// SIMATIC STEP 7 (V5.x) project zEn01_13_STEP7__PID-Temp
// program: Step controller
// program: Pulse controller
// program: Pulse control OB35, OB32
// program: Pulse control OB35, OB1
// program: Continuous controller

SYMBOL_TABLE
"DB_TCONT_S"	DB 59	FB 59
"DB_PROC_S"	DB 101	FB 101
"TCONT_S"	FB 59	FB 59	// temperature PID step controller
"PROC_S"	FB 101	FB 101
"CYC_INT5"	OB 35	OB 35
"COMPLETE_RESTART"	OB 100	OB 100
"VAT_LoopControlS"	VAT 1	
END_SYMBOL_TABLE

// FB 59: know-how protected block, not included

// FB 101: know-how protected block, not included

DATA_BLOCK "DB_TCONT_S"	// DB 59
VERSION : 0.0
"TCONT_S"
BEGIN
END_DATA_BLOCK

DATA_BLOCK "DB_PROC_S"	// DB 101
VERSION : 0.0
"PROC_S"
BEGIN
END_DATA_BLOCK

ORGANIZATION_BLOCK "CYC_INT5"	// OB 35
TITLE = "Cyclic Interrupt"
VERSION : 0.1
VAR_TEMP
  OB35_EV_CLASS : BYTE ;	//Bits 0-3 = 1 (Coming event), Bits 4-7 = 1 (Event class 1)
  OB35_STRT_INF : BYTE ;	//16#36 (OB 35 has started)
  OB35_PRIORITY : BYTE ;	//11 (Priority of 1 is lowest)
  OB35_OB_NUMBR : BYTE ;	//35 (Organization block 35, OB35)
  OB35_RESERVED_1 : BYTE ;	//Reserved for system
  OB35_RESERVED_2 : BYTE ;	//Reserved for system
  OB35_PHASE_OFFSET : WORD ;	//Phase offset (msec)
  OB35_RESERVED_3 : INT ;	//Reserved for system
  OB35_EXC_FREQ : INT ;	//Frequency of execution (msec)
  OB35_DATE_TIME : DATE_AND_TIME ;	//Date and time OB35 started
END_VAR
BEGIN
NETWORK
TITLE =
//Call the controller and the simulated process
      CALL  "TCONT_S" , "DB_TCONT_S" (
           DIX 18.0                 := DB101.DBX 50.0,
           DIX 18.1                 := DB101.DBX 50.1);
      CALL  "PROC_S" , "DB_PROC_S" (
           DIX 0.0                  := DB59.DBX 20.0,
           DIX 0.1                  := DB59.DBX 20.1,
           DID 42                   := DB59.DBD 8);
END_ORGANIZATION_BLOCK

ORGANIZATION_BLOCK "COMPLETE_RESTART"	// OB 100
TITLE = "Complete Restart"
VERSION : 0.1
VAR_TEMP
  OB100_EV_CLASS : BYTE ;	//16#13, Event class 1, Entering event state, Event logged in diagnostic buffer
  OB100_STRTUP : BYTE ;	//16#81/82/83/84 Method of startup
  OB100_PRIORITY : BYTE ;	//27 (Priority of 1 is lowest)
  OB100_OB_NUMBR : BYTE ;	//100 (Organization block 100, OB100)
  OB100_RESERVED_1 : BYTE ;	//Reserved for system
  OB100_RESERVED_2 : BYTE ;	//Reserved for system
  OB100_STOP : WORD ;	//Event that caused CPU to stop (16#4xxx)
  OB100_STRT_INFO : DWORD ;	//Information on how system started
  OB100_DATE_TIME : DATE_AND_TIME ;	//Date and time OB100 started
END_VAR
BEGIN
NETWORK
TITLE =
      SET;
//Startup routine for the controller and process
      =     DB59.DBX 30.0;
      =     DB101.DBX 52.0;
//Switch the controller to manual mode 
      =     DB59.DBX 18.2;
      L     0.000000e+00;
      T     DB101.DBD 46;
END_ORGANIZATION_BLOCK

SYMBOL_TABLE
"DB_TCONT_CP"	DB 58	FB 58
"DB_PROC_C"	DB 100	FB 100
"TCONT_CP"	FB 58	FB 58	// temperature PID controller with pulse generator and self-tuning
"PROC_C"	FB 100	FB 100	// process for continuous PID control
"CYC_INT5"	OB 35	OB 35	// Cyclic Interrupt 5
"COMPLETE RESTART"	OB 100	OB 100	// Complete Restart
"VAT_LoopControlC"	VAT 1	
END_SYMBOL_TABLE

// FB 58: know-how protected block, not included

// FB 100: know-how protected block, not included

DATA_BLOCK "DB_TCONT_CP"	// DB 58
AUTHOR : SIMATIC
FAMILY : CONTROL
VERSION : 0.0
"TCONT_CP"
BEGIN
END_DATA_BLOCK

DATA_BLOCK "DB_PROC_C"	// DB 100
AUTHOR : SIMATIC
FAMILY : PROCESS
VERSION : 0.0
"PROC_C"
BEGIN
END_DATA_BLOCK

ORGANIZATION_BLOCK "CYC_INT5"	// OB 35
TITLE = "Cyclic Interrupt"
VERSION : 0.1
VAR_TEMP
  OB35_EV_CLASS : BYTE ;	//Bits 0-3 = 1 (Coming event), Bits 4-7 = 1 (Event class 1)
  OB35_STRT_INF : BYTE ;	//16#36 (OB 35 has started)
  OB35_PRIORITY : BYTE ;	//11 (Priority of 1 is lowest)
  OB35_OB_NUMBR : BYTE ;	//35 (Organization block 35, OB35)
  OB35_RESERVED_1 : BYTE ;	//Reserved for system
  OB35_RESERVED_2 : BYTE ;	//Reserved for system
  OB35_PHASE_OFFSET : WORD ;	//Phase offset (msec)
  OB35_RESERVED_3 : INT ;	//Reserved for system
  OB35_EXC_FREQ : INT ;	//Frequency of execution (msec)
  OB35_DATE_TIME : DATE_AND_TIME ;	//Date and time OB35 started
END_VAR
BEGIN
NETWORK
TITLE =
//Call the controller and the simulated process
      CALL  "TCONT_CP" , "DB_TCONT_CP";
      CALL  "PROC_C" , "DB_PROC_C" (
           DID 0                    := DB58.DBD 18,
           DID 32                   := DB58.DBD 0);
END_ORGANIZATION_BLOCK

ORGANIZATION_BLOCK "COMPLETE RESTART"	// OB 100
TITLE = "Complete Restart"
VERSION : 0.1
VAR_TEMP
  OB100_EV_CLASS : BYTE ;	//16#13, Event class 1, Entering event state, Event logged in diagnostic buffer
  OB100_STRTUP : BYTE ;	//16#81/82/83/84 Method of startup
  OB100_PRIORITY : BYTE ;	//27 (Priority of 1 is lowest)
  OB100_OB_NUMBR : BYTE ;	//100 (Organization block 100, OB100)
  OB100_RESERVED_1 : BYTE ;	//Reserved for system
  OB100_RESERVED_2 : BYTE ;	//Reserved for system
  OB100_STOP : WORD ;	//Event that caused CPU to stop (16#4xxx)
  OB100_STRT_INFO : DWORD ;	//Information on how system started
  OB100_DATE_TIME : DATE_AND_TIME ;	//Date and time OB100 started
END_VAR
BEGIN
NETWORK
TITLE =
      SET;
//Startup routine for the controller and process
      =     DB58.DBX 42.0;
      =     DB100.DBX 36.0;
//Switch the controller to manual mode and output manipulated variable=0%
      =     DB58.DBX 42.1;
      L     0.000000e+00;
      T     DB58.DBD 38;
END_ORGANIZATION_BLOCK

SYMBOL_TABLE
"DB_TCONT_CP"	DB 58	FB 58
"DB_PROC_P"	DB 102	FB 102
"TCONT_CP"	FB 58	FB 58	// temperature PID controller with pulse generator and self-tuning
"PROC_P"	FB 102	FB 102	// process for puls control
"CYCL_EXC"	OB 1	OB 1	// Cycle Execution
"CYC_INT5"	OB 35	OB 35	// Cyclic Interrupt 5
"COMPLETE RESTART"	OB 100	OB 100	// Complete Restart
"VAT_LoopControl"	VAT 1	
END_SYMBOL_TABLE

// FB 58: know-how protected block, not included

// FB 102: know-how protected block, not included

DATA_BLOCK "DB_TCONT_CP"	// DB 58
AUTHOR : SIMATIC
FAMILY : CONTROL
VERSION : 0.0
"TCONT_CP"
BEGIN
END_DATA_BLOCK

DATA_BLOCK "DB_PROC_P"	// DB 102
AUTHOR : SIMATIC
FAMILY : PROCESS
VERSION : 0.0
"PROC_P"
BEGIN
END_DATA_BLOCK

ORGANIZATION_BLOCK "CYCL_EXC"	// OB 1
TITLE = "Main Program Sweep (Cycle)"
VERSION : 0.1
VAR_TEMP
  OB1_EV_CLASS : BYTE ;	//Bits 0-3 = 1 (Coming event), Bits 4-7 = 1 (Event class 1)
  OB1_SCAN_1 : BYTE ;	//1 (Cold restart scan 1 of OB 1), 3 (Scan 2-n of OB 1)
  OB1_PRIORITY : BYTE ;	//1 (Priority of 1 is lowest)
  OB1_OB_NUMBR : BYTE ;	//1 (Organization block 1, OB1)
  OB1_RESERVED_1 : BYTE ;	//Reserved for system
  OB1_RESERVED_2 : BYTE ;	//Reserved for system
  OB1_PREV_CYCLE : INT ;	//Cycle time of previous OB1 scan (milliseconds)
  OB1_MIN_CYCLE : INT ;	//Minimum cycle time of OB1 (milliseconds)
  OB1_MAX_CYCLE : INT ;	//Maximum cycle time of OB1 (milliseconds)
  OB1_DATE_TIME : DATE_AND_TIME ;	//Date and time OB1 started
END_VAR
BEGIN
NETWORK
TITLE =
//Call the controller
      A     DB58.DBX 24.3;
      JCN   M001;
      CALL  "TCONT_CP" , "DB_TCONT_CP" (
           DIW 12                   := 1);
M001: NOP   0;
END_ORGANIZATION_BLOCK

ORGANIZATION_BLOCK "CYC_INT5"	// OB 35
TITLE = "Cyclic Interrupt"
VERSION : 0.1
VAR_TEMP
  OB35_EV_CLASS : BYTE ;	//Bits 0-3 = 1 (Coming event), Bits 4-7 = 1 (Event class 1)
  OB35_STRT_INF : BYTE ;	//16#36 (OB 35 has started)
  OB35_PRIORITY : BYTE ;	//11 (Priority of 1 is lowest)
  OB35_OB_NUMBR : BYTE ;	//35 (Organization block 35, OB35)
  OB35_RESERVED_1 : BYTE ;	//Reserved for system
  OB35_RESERVED_2 : BYTE ;	//Reserved for system
  OB35_PHASE_OFFSET : WORD ;	//Phase offset (msec)
  OB35_RESERVED_3 : INT ;	//Reserved for system
  OB35_EXC_FREQ : INT ;	//Frequency of execution (msec)
  OB35_DATE_TIME : DATE_AND_TIME ;	//Date and time OB35 started
END_VAR
BEGIN
NETWORK
TITLE =
//Call the controller and the simulated process
      CALL  "TCONT_CP" , "DB_TCONT_CP" (
           DIW 12                   := 2);
      CALL  "PROC_P" , "DB_PROC_P" (
           DIX 0.0                  := DB58.DBX 24.0,
           DID 30                   := DB58.DBD 0);
END_ORGANIZATION_BLOCK

ORGANIZATION_BLOCK "COMPLETE RESTART"	// OB 100
TITLE = "Complete Restart"
VERSION : 0.1
VAR_TEMP
  OB100_EV_CLASS : BYTE ;	//16#13, Event class 1, Entering event state, Event logged in diagnostic buffer
  OB100_STRTUP : BYTE ;	//16#81/82/83/84 Method of startup
  OB100_PRIORITY : BYTE ;	//27 (Priority of 1 is lowest)
  OB100_OB_NUMBR : BYTE ;	//100 (Organization block 100, OB100)
  OB100_RESERVED_1 : BYTE ;	//Reserved for system
  OB100_RESERVED_2 : BYTE ;	//Reserved for system
  OB100_STOP : WORD ;	//Event that caused CPU to stop (16#4xxx)
  OB100_STRT_INFO : DWORD ;	//Information on how system started
  OB100_DATE_TIME : DATE_AND_TIME ;	//Date and time OB100 started
END_VAR
BEGIN
NETWORK
TITLE =
      SET;
//Startup routine for the controller and process
      =     DB58.DBX 42.0;
      =     DB102.DBX 34.0;
//Switch the controller to manual mode and output manipulated variable=0%
      =     DB58.DBX 42.1;
      L     0.000000e+00;
      T     DB58.DBD 38;
//Call mode of the pulse controller
      S     DB58.DBX 90.2;
END_ORGANIZATION_BLOCK

SYMBOL_TABLE
"DB_TCONT_CP"	DB 58	FB 58
"DB_PROC_P"	DB 102	FB 102
"TCONT_CP"	FB 58	FB 58	// temperature PID controller with pulse generator and self-tuning
"PROC_P"	FB 102	FB 102	// process for puls control
"CYCL_OB32"	OB 32	OB 32	// Cycle Execution
"CYC_OB35"	OB 35	OB 35	// Cyclic Interrupt 5
"COMPLETE RESTART"	OB 100	OB 100	// Complete Restart
"VAT_LoopControl"	VAT 1	
END_SYMBOL_TABLE

// FB 58: know-how protected block, not included

// FB 102: know-how protected block, not included

DATA_BLOCK "DB_TCONT_CP"	// DB 58
AUTHOR : SIMATIC
FAMILY : CONTROL
VERSION : 0.0
"TCONT_CP"
BEGIN
END_DATA_BLOCK

DATA_BLOCK "DB_PROC_P"	// DB 102
AUTHOR : SIMATIC
FAMILY : PROCESS
VERSION : 0.0
"PROC_P"
BEGIN
END_DATA_BLOCK

ORGANIZATION_BLOCK "CYCL_OB32"	// OB 32
TITLE = "Cyclic Interrupt"
VERSION : 0.1
VAR_TEMP
  OB32_EV_CLASS : BYTE ;	//Bits 0-3 = 1 (Coming event), Bits 4-7 = 1 (Event class 1)
  OB32_STRT_INF : BYTE ;	//16#33 (OB 32 has started)
  OB32_PRIORITY : BYTE ;	//Priority of OB Execution
  OB32_OB_NUMBR : BYTE ;	//32 (Organization block 32, OB32)
  OB32_RESERVED_1 : BYTE ;	//Reserved for system
  OB32_RESERVED_2 : BYTE ;	//Reserved for system
  OB32_PHS_OFFSET : INT ;	//Phase offset (integer, milliseconds)
  OB32_RESERVED_3 : INT ;	//Reserved for system
  OB32_EXC_FREQ : INT ;	//Frequency of execution (msec)
  OB32_DATE_TIME : DATE_AND_TIME ;	//Date and time OB32 started
END_VAR
BEGIN
NETWORK
TITLE =
//Call the controller
      CALL  "TCONT_CP" , "DB_TCONT_CP" (
           DIW 12                   := 3);
END_ORGANIZATION_BLOCK

ORGANIZATION_BLOCK "CYC_OB35"	// OB 35
TITLE = "Cyclic Interrupt"
VERSION : 0.1
VAR_TEMP
  OB35_EV_CLASS : BYTE ;	//Bits 0-3 = 1 (Coming event), Bits 4-7 = 1 (Event class 1)
  OB35_STRT_INF : BYTE ;	//16#36 (OB 35 has started)
  OB35_PRIORITY : BYTE ;	//11 (Priority of 1 is lowest)
  OB35_OB_NUMBR : BYTE ;	//35 (Organization block 35, OB35)
  OB35_RESERVED_1 : BYTE ;	//Reserved for system
  OB35_RESERVED_2 : BYTE ;	//Reserved for system
  OB35_PHASE_OFFSET : WORD ;	//Phase offset (msec)
  OB35_RESERVED_3 : INT ;	//Reserved for system
  OB35_EXC_FREQ : INT ;	//Frequency of execution (msec)
  OB35_DATE_TIME : DATE_AND_TIME ;	//Date and time OB35 started
END_VAR
BEGIN
NETWORK
TITLE =
//Call the pulse generator of controller and the simulated process
      CALL  "TCONT_CP" , "DB_TCONT_CP" (
           DIW 12                   := 2);
      CALL  "PROC_P" , "DB_PROC_P" (
           DIX 0.0                  := DB58.DBX 24.0,
           DID 30                   := DB58.DBD 0);
END_ORGANIZATION_BLOCK

ORGANIZATION_BLOCK "COMPLETE RESTART"	// OB 100
TITLE = "Complete Restart"
VERSION : 0.1
VAR_TEMP
  OB100_EV_CLASS : BYTE ;	//16#13, Event class 1, Entering event state, Event logged in diagnostic buffer
  OB100_STRTUP : BYTE ;	//16#81/82/83/84 Method of startup
  OB100_PRIORITY : BYTE ;	//27 (Priority of 1 is lowest)
  OB100_OB_NUMBR : BYTE ;	//100 (Organization block 100, OB100)
  OB100_RESERVED_1 : BYTE ;	//Reserved for system
  OB100_RESERVED_2 : BYTE ;	//Reserved for system
  OB100_STOP : WORD ;	//Event that caused CPU to stop (16#4xxx)
  OB100_STRT_INFO : DWORD ;	//Information on how system started
  OB100_DATE_TIME : DATE_AND_TIME ;	//Date and time OB100 started
END_VAR
BEGIN
NETWORK
TITLE =
      SET;
//Startup routine for the controller and process
      =     DB58.DBX 42.0;
      =     DB102.DBX 34.0;
//Switch the controller to manual mode and output manipulated variable=0%
      =     DB58.DBX 42.1;
      L     0.000000e+00;
      T     DB58.DBD 38;
//Call mode of the pulse controller
      S     DB58.DBX 90.2;
END_ORGANIZATION_BLOCK

SYMBOL_TABLE
"DB_TCONT_CP"	DB 58	FB 58
"DB_PROC_P"	DB 102	FB 102
"TCONT_CP"	FB 58	FB 58	// temperature PID controller with pulse generator and self-tuning
"PROC_P"	FB 102	FB 102	// process for puls control
"CYC_INT5"	OB 35	OB 35	// Cyclic Interrupt 5
"COMPLETE RESTART"	OB 100	OB 100	// Complete Restart
"VAT_LoopControl"	VAT 1	
"VAT_StructPar"	VAT 2	
END_SYMBOL_TABLE

// FB 58: know-how protected block, not included

// FB 102: know-how protected block, not included

DATA_BLOCK "DB_TCONT_CP"	// DB 58
AUTHOR : SIMATIC
FAMILY : CONTROL
VERSION : 0.0
"TCONT_CP"
BEGIN
END_DATA_BLOCK

DATA_BLOCK "DB_PROC_P"	// DB 102
AUTHOR : SIMATIC
FAMILY : PROCESS
VERSION : 0.0
"PROC_P"
BEGIN
END_DATA_BLOCK

ORGANIZATION_BLOCK "CYC_INT5"	// OB 35
TITLE = "Cyclic Interrupt"
VERSION : 0.1
VAR_TEMP
  OB35_EV_CLASS : BYTE ;	//Bits 0-3 = 1 (Coming event), Bits 4-7 = 1 (Event class 1)
  OB35_STRT_INF : BYTE ;	//16#36 (OB 35 has started)
  OB35_PRIORITY : BYTE ;	//11 (Priority of 1 is lowest)
  OB35_OB_NUMBR : BYTE ;	//35 (Organization block 35, OB35)
  OB35_RESERVED_1 : BYTE ;	//Reserved for system
  OB35_RESERVED_2 : BYTE ;	//Reserved for system
  OB35_PHASE_OFFSET : WORD ;	//Phase offset (msec)
  OB35_RESERVED_3 : INT ;	//Reserved for system
  OB35_EXC_FREQ : INT ;	//Frequency of execution (msec)
  OB35_DATE_TIME : DATE_AND_TIME ;	//Date and time OB35 started
END_VAR
BEGIN
NETWORK
TITLE =
//Call the controller and the simulated process
      CALL  "TCONT_CP" , "DB_TCONT_CP";
      CALL  "PROC_P" , "DB_PROC_P" (
           DIX 0.0                  := DB58.DBX 24.0,
           DID 30                   := DB58.DBD 0);
END_ORGANIZATION_BLOCK

ORGANIZATION_BLOCK "COMPLETE RESTART"	// OB 100
TITLE = "Complete Restart"
VERSION : 0.1
VAR_TEMP
  OB100_EV_CLASS : BYTE ;	//16#13, Event class 1, Entering event state, Event logged in diagnostic buffer
  OB100_STRTUP : BYTE ;	//16#81/82/83/84 Method of startup
  OB100_PRIORITY : BYTE ;	//27 (Priority of 1 is lowest)
  OB100_OB_NUMBR : BYTE ;	//100 (Organization block 100, OB100)
  OB100_RESERVED_1 : BYTE ;	//Reserved for system
  OB100_RESERVED_2 : BYTE ;	//Reserved for system
  OB100_STOP : WORD ;	//Event that caused CPU to stop (16#4xxx)
  OB100_STRT_INFO : DWORD ;	//Information on how system started
  OB100_DATE_TIME : DATE_AND_TIME ;	//Date and time OB100 started
END_VAR
BEGIN
NETWORK
TITLE =
      SET;
//Startup routine for the controller and process
      =     DB58.DBX 42.0;
      =     DB102.DBX 34.0;
//Switch the controller to manual mode and output manipulated variable=0%
      =     DB58.DBX 42.1;
      L     0.000000e+00;
      T     DB58.DBD 38;
//Call mode of the pulse controller
      L     0;
      T     DB58.DBW 12;
      S     DB58.DBX 90.2;
END_ORGANIZATION_BLOCK
